TYPE ST_Identity_PK1_OUT2 :
STRUCT
	ID	:STRING;
	ReadQuality:STRING;
END_STRUCT
END_TYPE

(* stored: Version 1.1.0.1, ProductVersion 3.1.4024.13
   DUT ST_Identity_PK1_OUT2: Id {c820eaab-ffd5-4458-a872-21d84738442e} *)
